// TIA Portal project "HW-setup-tcp1" (V14)

(* hardware
DEVICE "ET 200S station_1"  ET 200S station
   slot 0: "Rack_0"  Rail
   slot 2: "PLC_1"  IM151-8 CPU  6ES7 151-8AB00-0AB0  V2.7
      slot 1: "PROFINET interface_1"  PN-IO
         slot 1: "Port_1"  Port
         slot 2: "Port_2"  Port
         slot 3: "Port_3"  Port
   slot 4: "PM-E 24VDC_1"  PM-E 24VDC  6ES7 138-4CA01-0AA0
   slot 5: "8DO x 24VDC / 0.5A_1"  8DO x 24VDC / 0.5A  6ES7 132-4BF00-0AA0
   slot 6: "8DO x 24VDC / 0.5A_2"  8DO x 24VDC / 0.5A  6ES7 132-4BF00-0AA0
   slot 7: "8DI x 24VDC_1"  8DI x 24VDC  6ES7 131-4BF00-0AA0
   slot 8: "8DI x 24VDC_2"  8DI x 24VDC  6ES7 131-4BF00-0AA0
   slot 9: "8DI x 24VDC_3"  8DI x 24VDC  6ES7 131-4BF00-0AA0
   slot 10: "2AI x U ST_1"  2AI x U ST  6ES7 134-4FB01-0AB0
   slot 11: "2AI x U ST_2"  2AI x U ST  6ES7 134-4FB01-0AB0
   slot 12: "2AO x U ST_1"  2AO x U ST  6ES7 135-4FB01-0AB0
*)

// ===== PLC "PLC_1"  IM151-8 CPU =====

VAR_GLOBAL   // PLC tag table "IO"
   "DQ1" AT %QB1 : Byte;
   "DQ2" AT %QB2 : Byte;
   "DI1" AT %IB3 : Byte;
   "DI2" AT %IB4 : Byte;
   "DI3" AT %IB5 : Byte;
   "AI1-1" AT %IW352 : Int;
   "AI1-2" AT %IW354 : Int;
   "AI2-1" AT %IW356 : Int;
   "AI2-2" AT %IW358 : Int;
   "AQ1" AT %QW384 : Int;
   "AQ2" AT %QW386 : Int;
   "DQ1-1" AT %Q1.0 : Bool;
   "DQ1-2" AT %Q1.1 : Bool;
   "DQ1-3" AT %Q1.2 : Bool;
   "DQ1-4" AT %Q1.3 : Bool;
   "DQ1-5" AT %Q1.4 : Bool;
   "DQ1-6" AT %Q1.5 : Bool;
   "DQ1-7" AT %Q1.6 : Bool;
   "DQ1-8" AT %Q1.7 : Bool;
   "DI1-1" AT %I3.0 : Bool;
   "DI1-2" AT %I3.1 : Bool;
   "DI1-3" AT %I3.2 : Bool;
   "DI1-4" AT %I3.3 : Bool;
   "DI1-5" AT %I3.4 : Bool;
   "DI1-6" AT %I3.5 : Bool;
   "DI1-7" AT %I3.6 : Bool;
   "DI1-8" AT %I3.7 : Bool;
END_VAR

VAR_GLOBAL   // PLC tag table "M"
   "pot1" AT %MD10 : Real;
   "pot2" AT %MD14 : Real;
   "alwaysFalse" AT %M20.0 : Bool;
   "alwaysTrue" AT %M20.1 : Bool;
END_VAR

DATA_BLOCK "Diagnostics"   // DB1
{ S7_Optimized_Access := 'FALSE' }
VERSION : 0.1
   VAR
      scalePot1_retVal : Word;
      scalePot2_retVal : Word;
   END_VAR
BEGIN
END_DATA_BLOCK

FUNCTION_BLOCK "tcp"   // FB1, SCL
{ S7_Optimized_Access := 'FALSE' }
VERSION : 0.1
   VAR_INPUT
      enCom : Bool;
      enSend : Bool;
      enRcv : Bool;
      ID : Word;
   END_VAR
   VAR
      TCON_INST : TCON;
   END_VAR
   VAR_TEMP
      TCON_BUSY : Bool;
      TCON_DONE : Bool;
      TCON_ERROR : Bool;
      TCON_STATUS : Word;
   END_VAR
BEGIN
   #TCON_INST(REQ :=#enCom,
              ID :=#ID,
              CONNECT := P#DB2.DBX0.0 byte 64,
              BUSY =>#TCON_BUSY,
              DONE =>#TCON_DONE,
              ERROR =>#TCON_ERROR,
              STATUS =>#TCON_STATUS);
END_FUNCTION_BLOCK

FUNCTION "DigitalTest" : Void   // FC1, SCL
{ S7_Optimized_Access := 'FALSE' }
VERSION : 0.1
   VAR_INPUT
      in1 : Bool;
      in2 : Bool;
      in3 : Bool;
      in4 : Bool;
      in5 : Bool;
      in6 : Bool;
      in7 : Bool;
      in8 : Bool;
   END_VAR
   VAR_OUTPUT
      out1 : Bool;
      out2 : Bool;
      out3 : Bool;
      out4 : Bool;
      out5 : Bool;
      out6 : Bool;
      out7 : Bool;
      out8 : Bool;
   END_VAR
BEGIN
   #out1 := #in1;
   #out2 := #in2;
   #out3 := #in3;
   #out4 := #in4;
   #out5 := #in5;
   #out6 := #in6;
   #out7 := #in7;
   #out8 := #in8;
END_FUNCTION

ORGANIZATION_BLOCK "Main"   // OB1, LAD
TITLE = "Main Program Sweep (Cycle)"
{ S7_Optimized_Access := 'FALSE' }
VERSION : 0.1
   VAR_TEMP
      OB1_EV_CLASS : Byte;   // Bits 0-3 = 1 (Coming event), Bits 4-7 = 1 (Event class 1)
      OB1_SCAN_1 : Byte;   // 1 (Cold restart scan 1 of OB 1), 3 (Scan 2-n of OB 1)
      OB1_PRIORITY : Byte;   // Priority of OB Execution
      OB1_OB_NUMBR : Byte;   // 1 (Organization block 1, OB1)
      OB1_RESERVED_1 : Byte;   // Reserved for system
      OB1_RESERVED_2 : Byte;   // Reserved for system
      OB1_PREV_CYCLE : Int;   // Cycle time of previous OB1 scan (milliseconds)
      OB1_MIN_CYCLE : Int;   // Minimum cycle time of OB1 (milliseconds)
      OB1_MAX_CYCLE : Int;   // Maximum cycle time of OB1 (milliseconds)
      OB1_DATE_TIME : Date_And_Time;   // Date and time OB1 started
   END_VAR
BEGIN

REGION Network 1: Test digital IO
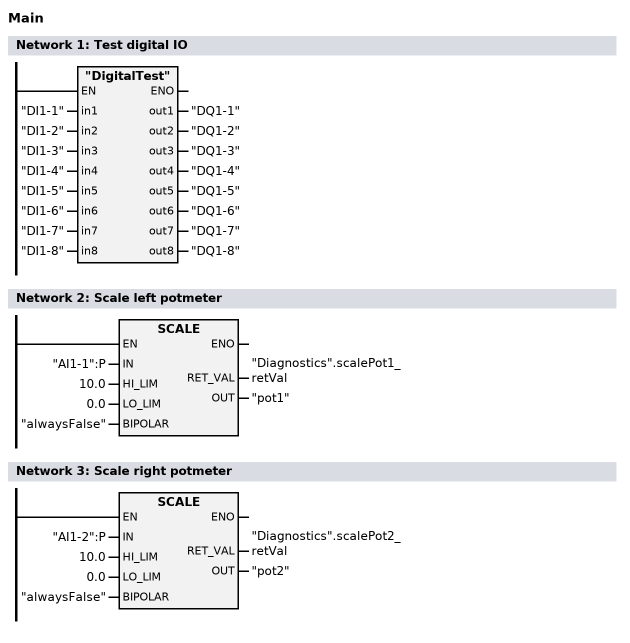
   RUNG wire#powerrail
      "DigitalTest"(in1 := "DI1-1", in2 := "DI1-2", in3 := "DI1-3", in4 := "DI1-4", in5 := "DI1-5", in6 := "DI1-6", in7 := "DI1-7", in8 := "DI1-8", out1 => "DQ1-1", out2 => "DQ1-2", out3 => "DQ1-3", out4 => "DQ1-4", out5 => "DQ1-5", out6 => "DQ1-6", out7 => "DQ1-7", out8 => "DQ1-8")
   END_RUNG
   // the same network as SCL:
   "DigitalTest"(in1 := "DI1-1",
                 in2 := "DI1-2",
                 in3 := "DI1-3",
                 in4 := "DI1-4",
                 in5 := "DI1-5",
                 in6 := "DI1-6",
                 in7 := "DI1-7",
                 in8 := "DI1-8",
                 out1 => "DQ1-1",
                 out2 => "DQ1-2",
                 out3 => "DQ1-3",
                 out4 => "DQ1-4",
                 out5 => "DQ1-5",
                 out6 => "DQ1-6",
                 out7 => "DQ1-7",
                 out8 => "DQ1-8");
END_REGION

REGION Network 2: Scale left potmeter
   "Diagnostics".scalePot1_retVal := SCALE(IN := "AI1-1":P,
                           HI_LIM := 10.0,
                           LO_LIM := 0.0,
                           BIPOLAR := "alwaysFalse",
                           OUT => "pot1");
END_REGION

REGION Network 3: Scale right potmeter
   "Diagnostics".scalePot2_retVal := SCALE(IN := "AI1-2":P,
                           HI_LIM := 10.0,
                           LO_LIM := 0.0,
                           BIPOLAR := "alwaysFalse",
                           OUT => "pot2");
END_REGION
END_ORGANIZATION_BLOCK

ORGANIZATION_BLOCK "COMPLETE RESTART"   // OB100, SCL
TITLE = "Complete Restart"
{ S7_Optimized_Access := 'FALSE' }
VERSION : 0.1
   VAR_TEMP
      OB100_EV_CLASS : Byte;   // 16#13, Event class 1, Entering event state, Event logged in diagnostic buffer
      OB100_STRTUP : Byte;   // 16#81/82/83/84 Method of startup
      OB100_PRIORITY : Byte;   // Priority of OB Execution
      OB100_OB_NUMBR : Byte;   // 100 (Organization block 100, OB100)
      OB100_RESERVED_1 : Byte;   // Reserved for system
      OB100_RESERVED_2 : Byte;   // Reserved for system
      OB100_STOP : Word;   // Event that caused CPU to stop (16#4xxx)
      OB100_STRT_INFO : DWord;   // Information on how system started
      OB100_DATE_TIME : Date_And_Time;   // Date and time OB100 started
   END_VAR
BEGIN
   "alwaysFalse" := "alwaysFalse" AND NOT "alwaysFalse";
   "alwaysTrue" := "alwaysTrue" OR NOT "alwaysTrue";
END_ORGANIZATION_BLOCK